Universal Robots PolyScope program: positionTest.urp

Program positionTest (installation=default_3 directory=/programs/usbdisk createdIn=5.18.0 lastSavedIn=5.18.0 robotSerialNumber=20245388888)
Calibrated DH parameters: a=[0, -0.24355, -0.2132, 0, 0, 0]; d=[0.15185, 0, 0, 0.13105, 0.08535, 0.0921]; alpha=[1.570796, 0, 0, 1.570796, -1.570796, 0]; deltaTheta=[0, 0, 0, 0, 0, 0]
InitVariablesNode
Robot Program (runOnlyOnce=false)
  MoveL speed 250 mm/s, acceleration 1200 mm/s^2 (useActiveTCP=true optimoveEnabled=true optiMovePercentage=30) feature=Base
    Waypoint Waypoint_1: TCP in base x=-164.146 y=128.516 z=466.6 mm, rx=-0.0259 ry=0.034 rz=1.6093 rad; joints [182.133, -177.642, 87.162, 0.813, 87.83, 0.08] deg
